		(*******************************************************************************
		  Modify error 
		********************************************************************************)
		E_ITC_MsgTypeConv.E_ERROR_REQUEST:
			M_ITC_ERQ(meChannelSrc := meChannelSrc, mpData := mpData, mLen := mLen);

	ELSE
		// Unknown ITC message type received
		DebugMsg := CONCAT('Subsystem emulation unknown ITC Message type: ', INT_TO_STRING(SubsystemBase.eITC_MsgType));
		fbDebugMsg.M_SendErrorMsg(DebugMsg);
	END_CASE

END_IF
END_METHOD

METHOD M_UpdateRealObjectData
(**************************************************************************************
 * 	Application		:	BoxControl Framework
 *	Revision		:	$Revision: 404529 $
 *	Revision date	:	$Date: 2018-04-23 08:21:38 +0200 (Mo., 23 Apr 2018) $
 *	Last changed by	:	$Author: b7bolm $
 *	URL				:	$URL: http://almscdc.swisslog.com/repo/SWPD/Development/BoxControlFramework/20_Release/trunk/01_Software/BCF/BCF/JumpStart/20_Product/11_Emu/15_Subsystem/10_Lib/10_Conv/FB_SubsystemConvEmulation.TcPOU $
 *
 *	Purpose			:	This methode gets always the current values of the real object
 *
 * ------------------------------------------------------------------------------------
 *	Copyright Swisslog [IP AG], Switzerland. All rights reserved.
 * 
 * ------------------------------------------------------------------------------------
 *	
 * 	Revision History: 
 *
 * 	VERSION			DATE			INITIALS			DESCRIPTION
 *	0.1				01.01.2001		swl					Example
 *
 **************************************************************************************)

IF __ISVALIDREF(SubsystemRegistry.rSubsystemData) THEN
	SubsystemBase.rSubsystemDataReal REF= SubsystemRegistry.rSubsystemData;
ELSE
	SubsystemBase.rSubsystemDataReal REF= SubsystemBase.SubsystemDataEmpty;
END_IF

IF __ISVALIDREF(SubsystemRegistry.rSubsystemInterface) THEN
	SubsystemBase.rSubsystemInterfaceReal REF= SubsystemRegistry.rSubsystemInterface;
ELSE
	SubsystemBase.rSubsystemInterfaceReal REF= SubsystemBase.SubsystemInterfaceEmpty;
END_IF

IF __ISVALIDREF(SubsystemRegistry.rSettingsSubsystem) THEN
	SubsystemBase.rSettingsSubsystemReal REF= SubsystemRegistry.rSettingsSubsystem;
ELSE
	SubsystemBase.rSettingsSubsystemReal REF= SubsystemBase.SettingsSubsystemEmpty;
END_IF
END_METHOD

END_FUNCTION_BLOCK

// ---- 20_Product/10_BCF/10_Base/11_Com/12_DebugMsg/FB_DebugMsgManager.TcPOU
{attribute 'reflection' := ''}
FUNCTION_BLOCK FB_DebugMsgManager
(**************************************************************************************
 * 	Application		:	BoxControl Framework
 *	Revision		:	$Revision: 404529 $
 *	Revision date	:	$Date: 2018-04-23 08:21:38 +0200 (Mo., 23 Apr 2018) $
 *	Last changed by	:	$Author: b7bolm $
 *	URL				:	$URL: http://almscdc.swisslog.com/repo/SWPD/Development/BoxControlFramework/20_Release/trunk/01_Software/BCF/BCF/JumpStart/20_Product/10_App/11_Com/10_Lib/FB_DebugMsgManager.TcPOU $
 *
 *	Purpose			:	Debug msg manager 
 *
 * ------------------------------------------------------------------------------------
 *	Copyright Swisslog [IP AG], Switzerland. All rights reserved.
 * 
 * ------------------------------------------------------------------------------------
 *	
 * 	Revision History: 
 *
 * VERSION DATE         INITIALS     DESCRIPTION
 * 0.0     DD.MM.YYYY   (name)       (explain customized modifications)
 *
 **************************************************************************************)
VAR_INPUT
	Config						: ST_CFG_DebugMsgManager;	// Configuration of debug msg manager
	//-----------------------------------------------------------------------------------
	EnableInfos					: BOOL		:= TRUE;		// Enables debug messages for infos
	EnableWarnings				: BOOL		:= TRUE;		// Enables debug messages for warnings
	EnableErrors				: BOOL		:= TRUE;		// Enables debug messages for errors
END_VAR
 
VAR
	DebugMsg					: T_MaxString; // String to compose the logmessage
	fbDebugMsg					: FB_DebugMsg; // Object Debug instance
	fbTCP_Driver				: FB_TCP_Driver; // Instance of a TCP/IP connection handler
	AddByteMessage				: ARRAY[1 .. MAX_MSG_LENGTH] OF BYTE; // Added byte message
	ReadByteMessage				: ARRAY[1 .. MAX_MSG_LENGTH] OF BYTE; // Read out message
	CollectedByteMessage		: ARRAY[1 .. MAX_MSG_LENGTH] OF BYTE; // Collected byte message
	SendBufferSpace				: ARRAY[1 .. MAX_BUFFER_SPACE] OF BYTE; // Space for send messages
	fbSendBuffer				: FB_MemRingBuffer; // Send buffer
	Header						: T_MaxString; // Collected header
	LastAddedMsg				: T_MaxString; // Debug message last added message
	LastSentMsg					: T_MaxString; // Debug message last sent
	WritePointer				: UDINT; // Counter for assembling byte stream
	NoError						: BOOL; // No error during operation
	DataReady					: BOOL; // Data ready to send
	Idx							: INT; // Index for iteration	
	RecvData					: ARRAY[1..10] OF BYTE; // Receive buffer
	fbFileHandler				: FB_TraceHandler(); 					// trace file handler
END_VAR

VAR CONSTANT
	MAX_MSG_LENGTH				: DINT := 30000; // Maximum byte length of a message
	MAX_BUFFER_SPACE			: DINT := 30000; // Allocated send buffer space
	MSG_PER_CYCLE				: INT := 5; // Maximum collected messages
	DEBUGMESSAGETYPELENGTH 		: INT := 20; // String length debug message type
END_VAR


// call file handler
fbFileHandler();

// Only handle all entries, if a connection is established
IF fbTCP_Driver.Connected THEN
	// Check if a message to send is available and the sending channel is free to send
	IF NOT fbTCP_Driver.SendBusy AND fbSendBuffer.nCount > 0 THEN
			
		// Initialize values
		MEMSET(destAddr := ADR(CollectedByteMessage), 0, SIZEOF(CollectedByteMessage));
		WritePointer := 0;
		DataReady := FALSE;
		(*
		In order to send efficiently, it will be tried to collect
		multiple messages to one TCP/IP stream.
		
		Generell it will be tried to collect everytime MSG_PER_CYCLE messages.
		After MSG_PER_CYCLE messages or if the added messages exeeds MAX_MSG_LENGTH, 
		no more messages will be added.
		*)
		FOR Idx := 1 TO MSG_PER_CYCLE DO
			// If send buffer consists of unsent messages
			IF fbSendBuffer.nCount > 0 THEN
				// Clear byte stream
				MEMSET(destAddr := ADR(ReadByteMessage), 0, SIZEOF(ReadByteMessage));
				
				// Read next message out of the buffer (But not remove)
				fbSendBuffer.A_GetHead(
					pBuffer := ADR(SendBufferSpace), 
					cbBuffer := SIZEOF(SendBufferSpace), 
					pRead := ADR(ReadByteMessage), 
					cbRead := SIZEOF(ReadByteMessage));
				
				// If read out was successfully
				IF fbSendBuffer.bOk THEN
					// Append source
					NoError := F_AssembleByteStream(
									pSrc := ADR(ReadByteMessage), 
									SrcLen := fbSendBuffer.cbReturn,
									pDest := ADR(CollectedByteMessage), 
									DestLen := SIZEOF(CollectedByteMessage),
									WritePointer := WritePointer);
					
					// if assembling was successful (Maybe the message was to long and therefore not adable
					IF NoError THEN
						// As a reason that the message could be assembled, remove from buffer
						fbSendBuffer.A_RemoveHead(
							pBuffer := ADR(SendBufferSpace), 
							cbBuffer := SIZEOF(SendBufferSpace), 
							pRead := ADR(ReadByteMessage), 
							cbRead := SIZEOF(ReadByteMessage));
							
						// Data assembled
						DataReady := TRUE;
					ELSE
						(*
						It was not possible to add MSG_PER_CYCLE messages.
						Already added messages exeeded MAX_MSG_LENGTH
						*)
						EXIT;
					END_IF	
				ELSE
					DebugMsg := CONCAT('CRITICAL Buffer read out. ReturnValue:', UDINT_TO_STRING(fbSendBuffer.cbReturn));
					fbDebugMsg.M_SendErrorMsg(DebugMsg);	
				END_IF
			ELSE
				// No further messages waiting
				EXIT;
			END_IF
		END_FOR
	
		// If data needs to be sent
		IF DataReady THEN
			// Send command
			fbTCP_Driver.M_Send(
				mpSendData	:= ADR(CollectedByteMessage),
				mSendDataLen:= WritePointer);
				
			// Store first 255 characters for debugging
			F_BlockCopy(
				pSrc:= ADR(CollectedByteMessage), 
				LenSrc:= WritePointer, 
				pDest:= ADR(LastSentMsg), 
				LenDest:= SIZEOF(LastSentMsg));
		END_IF
	END_IF
END_IF

// Cylic update of TCP/ IP driver
// Receive is not needed for debug messages, therefore no receive structure is allocated
// Call is at the end, to gain one cycle of a sending request
fbTCP_Driver(
	Config := Config.TCP_Driver, 
    pReceiveData := ADR(RecvData),
	ReceiveDataLen := SIZEOF(RecvData));

// file handler
{attribute 'monitoring' := 'call'}
PROPERTY PUBLIC FileHandler : I_TraceHandler
GET
FileHandler:= fbFileHandler;
END_GET
END_PROPERTY

{attribute 'object_name' := 'M_SendMessage'}
METHOD M_SendMessage : BOOL
(**************************************************************************************
 * 	Application		:	BoxControl Framework
 *	Revision		:	$Revision: 404529 $
 *	Revision date	:	$Date: 2018-04-23 08:21:38 +0200 (Mo., 23 Apr 2018) $
 *	Last changed by	:	$Author: b7bolm $
 *	URL				:	$URL: http://almscdc.swisslog.com/repo/SWPD/Development/BoxControlFramework/20_Release/trunk/01_Software/BCF/BCF/JumpStart/20_Product/10_App/11_Com/10_Lib/FB_DebugMsgManager.TcPOU $
 *
 *	Purpose			:	Send  message
 *
 * ------------------------------------------------------------------------------------
 *	Copyright Swisslog [IP AG], Switzerland. All rights reserved.
 * 
 * ------------------------------------------------------------------------------------
 *	
 * 	Revision History: 
 *
 * 	VERSION			DATE			INITIALS			DESCRIPTION
 *	0.1				01.01.2001		swl					Example
 *
 **************************************************************************************)
VAR_INPUT
	meMessageType		: E_DebugMsgType;
	mDebugSource		: STRING(DEBUGSOURCELENGTH);
	mpMsgData			: PVOID; // Address to the send data storage
	mMsgDataLen			: UDINT; // Data length which need to be sent
END_VAR

VAR
	mString				:STRING(10); // Temp String
END_VAR

// forward to file handler
fbFileHandler.Put(MsgType :=     meMessageType,
                  Instance:= ADR(mDebugSource),
                  Text    :=     mpMsgData);


// Translate to string
CASE meMessageType OF
E_DebugMsgType.INFO:		IF NOT EnableInfos		THEN  M_SendMessage:= FALSE;  RETURN;  END_IF
E_DebugMsgType.WARNING:		IF NOT EnableWarnings	THEN  M_SendMessage:= FALSE;  RETURN;  END_IF
E_DebugMsgType.ERROR:		IF NOT EnableErrors		THEN  M_SendMessage:= FALSE;  RETURN;  END_IF
ELSE						meMessageType:= E_DebugMsgType.ERROR;
END_CASE


// Reset
MEMSET(destAddr := ADR(AddByteMessage), 0, SIZEOF(AddByteMessage));
WritePointer := 0;

Header := CONCAT('<', TimeStampString);
Header := CONCAT(Header, ', ');
Header := CONCAT(Header, TO_STRING(meMessageType));
Header := CONCAT(Header, ', System: ');
Header := CONCAT(Header, INT_TO_STRING(Config.SystemNumber));
Header := CONCAT(Header, ', ');
Header := CONCAT(Header, mDebugSource);
Header := CONCAT(Header, ', ');

// Append header
F_AssembleByteStream(
	pSrc := ADR(Header),
	SrcLen := INT_TO_UDINT(LEN(Header)),
	pDest := ADR(AddByteMessage), 
	DestLen := SIZEOF(AddByteMessage),
	WritePointer := WritePointer);

// Append message
F_BlockCopy(
	pSrc := mpMsgData,
	LenSrc := mMsgDataLen, 
	pDest := ADR(AddByteMessage) + WritePointer,
	LenDest := SIZEOF(AddByteMessage) - WritePointer);

// Update pointer
WritePointer := WritePointer + mMsgDataLen;

// Append end sign + Line feed
mString := '>$0A';

F_AssembleByteStream(
	pSrc := ADR(mString), 
	SrcLen := INT_TO_UDINT(LEN(mString)),
	pDest := ADR(AddByteMessage), 
	DestLen := SIZEOF(AddByteMessage),
	WritePointer := WritePointer);


// Add to byte buffer in order to release caller
fbSendBuffer.A_AddTail(
	pBuffer := ADR(SendBufferSpace), 
	cbBuffer := SIZEOF(SendBufferSpace), 
	pWrite := ADR(AddByteMessage), 
	cbWrite := WritePointer);

IF NOT fbSendBuffer.bOk THEN
	// Remove oldest entry
	fbSendBuffer.A_RemoveHead(
		pBuffer := ADR(SendBufferSpace), 
		cbBuffer := SIZEOF(SendBufferSpace), 
		pRead := ADR(ReadByteMessage), 
		cbRead := SIZEOF(ReadByteMessage));

	// Add to byte buffer in order to release caller
	fbSendBuffer.A_AddTail(
		pBuffer := ADR(SendBufferSpace), 
		cbBuffer := SIZEOF(SendBufferSpace), 
		pWrite := ADR(AddByteMessage), 
		cbWrite := WritePointer);
END_IF

// Store first 255 characters for debugging
F_BlockCopy(
	pSrc:= ADR(AddByteMessage), 
	LenSrc:= WritePointer, 
	pDest:= ADR(LastAddedMsg), 
	LenDest:= SIZEOF(LastAddedMsg));
	
// Return result
M_SendMessage := fbSendBuffer.bOk;
END_METHOD

END_FUNCTION_BLOCK

// ---- 20_Product/30_Toolbox/11_Com/10_TCP_Driver/FB_TCP_Driver.TcPOU
///TCP / IP Driver - Handles a connection to one partner. Handles only one incoming and one outgoing message at once.
FUNCTION_BLOCK FB_TCP_Driver
(**************************************************************************************
* Application : BoxControl Framework 
* Revision date : $Date: 2020-10-16 11:02:56 +0200 (fre, 16 okt 2020) $
* Author : CDC
* ------------------------------------------------------------------------------------ 
* © Swisslog AG 
* Swisslog is not liable for any usage of this source code that is not agreed 
* on between Swisslog and the other party. The mandatory legal liability remains 
* unaffected. 
* ------------------------------------------------------------------------------------ 
* Project revision history: 
* 
* VERSION 	DATE 		INITIALS 	DESCRIPTION 
* 0.1 		12.10.2020 	swl. 		example
* 
**************************************************************************************)

VAR_INPUT
	Config						: ST_CFG_TcpDriver;
	pReceiveData				: PVOID; // Pointer to receive structure
	ReceiveDataLen				: UDINT; // Length of received structure (Maximum which could be received)

END_VAR

VAR_OUTPUT
	NewData						: BOOL; // New Data received	
	ReceivedBytes				: UDINT; // Amount of received bytes
	Connected					: BOOL; // Connected 
	
	ConnBusy					: BOOL; // Connection ongoing
	ConnError					: BOOL; // Error during connection
	ConnErrId					: UDINT; // Connection error code
		
	SendBusy					: BOOL; // Send ongoing status	
	SendError					: BOOL; // Send error
	SendErrId					: UDINT; // Sending error code
	
	RecvBusy					: BOOL; // Receive ongoing status
	RecvError					: BOOL; // Receive error
	RecvErrId					: UDINT; // Receive error code
END_VAR

VAR

	Init						: BOOL := FALSE; // Instance is initialized
	fbDebugMsg					: FB_DebugMsg; // Debug msg handler
	DebugMsg					: T_MAXSTRING; // Debug msg
	EnableSystemLog				: BOOL	:= FALSE;

	fbConnectClientServer		: FB_ClientServerConnection := (sSrvNetId := ''); // Tc library connect
	fbConnectServerClient		: FB_ServerClientConnection; // Tc library connect
	
	fbSocketSend				: FB_SocketSend := (sSrvNetID := '', tTimeout := DEFAULT_ADS_TIMEOUT); // Tc library send
	fbSocketReceive				: FB_SocketReceive := (sSrvNetID := '', tTimeout := DEFAULT_ADS_TIMEOUT); // Tc library recv
	hServer						: T_HSERVER; // Server connection handle 
	hSocket						: T_HSOCKET; // Connection socket
	
	// Send receive data
	RecvString					: T_MaxString; // String received for debugging
	SendString					: T_MaxString; // String send for debugging
	pSendData					: PVOID; // Address send structure
	SendDataLen					: UDINT; // Send data length
	
	// States	
	SocketState					: E_SocketConnectionState := eSOCKET_DISCONNECTED; // TCP/IP connection state 
	ConnState					: E_ConnStates; // Connection states
	SendState					: E_SendStates; // Sending states
	RecvState					: E_RecvStates; // Receive states

	SendTrigger					: BOOL; // New Data to Send
	RestartCom					: BOOL; // Close and reopen socket

	// Socket variables to accept and refuse a second server connection 
	fbConnectServer_ConRefuse	: FB_ServerClientConnection; // Establishes a connection 
	hSocket_ConRefuse			: T_HSOCKET; // Socket handle for this connection
	SocketState_ConRefuse		: E_SocketConnectionState := eSOCKET_DISCONNECTED; // Socket state

	ConnState_ConRefuse			: E_ConnStates; // Connection states; 

	fbSocketSend_ConRefuse		: FB_SocketSend := (sSrvNetID := '', tTimeout := DEFAULT_ADS_TIMEOUT); // Send function block
	MsgConnection_ConRefuse		: STRING := 'Connection refused'; // 

END_VAR

(**************************************************************************************
   		Initialize
***************************************************************************************)

M_Init(FALSE);

//  Server mode
IF Config.Server THEN
	// Call connection handling as server
	A_Server();
	
	// Reject additional incomming connection requests
	A_RejectCon();
	
// Client mode	
ELSE
	// Call connection handling as client
	A_Client();
END_IF

ACTION A_Client:
fbConnectClientServer(hSocket => hSocket);

// Connection states
CASE ConnState OF
	// Connection is idle 
	E_ConnStates.CONN_IDLE:
		Connected := FALSE;
		// If connection is enabled 
		IF Config.EnableConnection THEN
			// Poll connection for new client
			fbConnectClientServer( 	
						nMode			:= SEL( EnableSystemLog, 0, CONNECT_MODE_ENABLEDBG), // Enable/disable debug messages? 
						sRemoteHost 	:= Config.RemoteHost, 
						nRemotePort 	:= Config.RemotePort,
						bEnable			:= TRUE, 
						tReconnect		:= Config.ClientRetryInterval, // Retry connection after  ConnectionTimeout
						eState			=> SocketState );
						
			IF NOT fbConnectClientServer.bBusy THEN
				IF NOT fbConnectClientServer.bError THEN
					IF SocketState = eSOCKET_CONNECTED THEN  // We are connected 
											
						SendBusy 	:= FALSE;
						RecvBusy 	:= FALSE;
	
						Connected := TRUE;
						ConnState := E_ConnStates.CONN_RUNNING;
					END_IF
				END_IF
			END_IF				
		
		END_IF
		

	// Connection is established - execute sending and receive over the connection 
	E_ConnStates.CONN_RUNNING:
		// Send
		A_Send();
		// Recv
		A_Recv();

	
		// Should the connection need to be disabled or an error occours in the sending/receiving of data, deal with it 
		IF NOT Config.EnableConnection AND NOT fbSocketSend.bBusy AND NOT fbSocketReceive.bBusy OR RestartCom THEN
			RestartCom := FALSE;
			M_DebugSendInfoMsg('ConnState: CONN_CLOSE_START');
			ConnState := E_ConnStates.CONN_CLOSE;
			
		ELSIF SendError OR RecvError THEN
			SendError := FALSE;
			RecvError := FALSE;
			M_DebugSendInfoMsg('ConnState: CONN_ERROR');
			ConnState := E_ConnStates.CONN_ERROR;
		END_IF
		
	// Connections need to be closed 
	E_ConnStates.CONN_CLOSE:
		fbConnectClientServer( bEnable:= FALSE, eState => SocketState );
		IF SocketState = eSOCKET_DISCONNECTED THEN
			// Please wait some seconds and then try to connect again 
			Connected := FALSE;
			RecvState := E_RecvStates.RECV_IDLE;
			SendState := E_SendStates.SEND_IDLE;
			ConnState := E_ConnStates.CONN_IDLE;
		END_IF
		
	// Error detected in connection 
	E_ConnStates.CONN_ERROR:
		
		// If still connected
		IF Connected THEN
			// Close connection
			M_DebugSendInfoMsg('ConnState: CONN_CLOSE_START');
			ConnState := E_ConnStates.CONN_CLOSE;
		ELSE
			ConnBusy   := FALSE;
			// Switch to idle
			M_DebugSendInfoMsg('ConnState: CONN_IDLE');
			ConnState := E_ConnStates.CONN_IDLE;
		END_IF
END_CASE
END_ACTION

ACTION A_Recv:
// Receive states
CASE RecvState OF
	// Idle state - waiting for confirmation to enable receiving 
	E_RecvStates.RECV_IDLE:
		// If no new data are waiting to be removed and
		// a valid receive structure is available
		IF NOT NewData AND
           pReceiveData <> 0 AND 
           ReceiveDataLen > 0 THEN
			// Block receive channel
			RecvBusy := TRUE;
			
			// Call receive function block
			fbSocketReceive(
				hSocket  	:= hSocket,
				pDest	 	:= pReceiveData,
				cbLen	 	:= ReceiveDataLen,
				bExecute 	:= TRUE);
			
			// Reset variables
			RecvError := FALSE;
			RecvErrId := 0;
			ReceivedBytes := 0;
			MEMSET(ADR(RecvString), 0, SIZEOF(RecvString));
			
			// Switch to receive start
			RecvState := E_RecvStates.RECV_WAIT;
		
		END_IF
		
	// Receiving is active, wait for the function to complete 
	E_RecvStates.RECV_WAIT:
		// Reset
		fbSocketReceive(bExecute := FALSE);
		
		// If receiving is finished
		IF NOT fbSocketReceive.bBusy THEN
			// Reset
			RecvBusy := FALSE;	
		
			// If no error is occured
			IF NOT fbSocketReceive.bError THEN
				// Receive module has completed - analyse the message 
				IF (fbSocketReceive.nRecBytes > 0) THEN
					// Store received bytes 
					ReceivedBytes := fbSocketReceive.nRecBytes;
				
					// Copy first 255 signs for debug reason to RecvString
					F_BlockCopy(
						pSrc:= pReceiveData, 
						LenSrc:= ReceivedBytes, 
						pDest:= ADR(RecvString), 
						LenDest:= SIZEOF(RecvString));
						
					// Set new data ready
					NewData := TRUE;
				END_IF
				// Go to Idle
				RecvState := E_RecvStates.RECV_IDLE;
			ELSE
				// Error detected 
				RecvErrId := fbSocketReceive.nErrId;
				RecvState := E_RecvStates.RECV_ERROR;
			END_IF
		END_IF
		
	// Recv error state 
	E_RecvStates.RECV_ERROR:
		RecvBusy := FALSE;
		RecvError := TRUE;
		RecvState := E_RecvStates.RECV_IDLE;
END_CASE
END_ACTION

ACTION A_RejectCon:
(* -----------------------------------------------------------------------------
 	This code avoids addional connection as soon as a connection was established
 	It will accept any new incomming connection requests and will close it immediately
-------------------------------------------------------------------------------- *)

// Connection alreads established check for new incomming connection requests
IF ConnState <> E_ConnStates.CONN_IDLE THEN

	// Connection states
	CASE ConnState_ConRefuse OF
		// Connection is idle 
		E_ConnStates.CONN_IDLE:
			
			// If connection is enabled and not listening
			IF Config.EnableConnection THEN
				fbConnectServer_ConRefuse( 	eMode := eACCEPT_ALL, 
								tReconnect := Config.ServerRetryInterval, // Retry connection after  ConnectionTimeout
								bEnable := TRUE, 
								hServer := hServer, 
								hSocket => hSocket_ConRefuse, 
								eState => SocketState_ConRefuse );
								
				IF NOT fbConnectServer_ConRefuse.bBusy THEN
					IF NOT fbConnectServer_ConRefuse.bError THEN
						IF SocketState = eSOCKET_CONNECTED THEN(* We are connected *)
							ConnState_ConRefuse := E_ConnStates.CONN_RUNNING;
						END_IF
					END_IF
				END_IF
			END_IF
	
		// Socket is open and listening, process incoming connection requests from partner 
		E_ConnStates.CONN_RUNNING:
					
			// Start send action in same cycle
			MsgConnection_ConRefuse := 'Connection refused, already active Connection with IP = ';
			MsgConnection_ConRefuse := concat(MsgConnection_ConRefuse, fbConnectServerClient.hSocket.remoteAddr.sAddr);

			// Send the connection refused message to the client
			fbSocketSend_ConRefuse(
				hSocket  	:= hSocket_ConRefuse,
				pSrc     	:= ADR(MsgConnection_ConRefuse),
				cbLen    	:= SIZEOF(MsgConnection_ConRefuse),
				bExecute 	:= TRUE);
					
					
			// Continue to wait, until the FB_SocketSend instance has finished and close the connection
			IF NOT fbSocketSend_ConRefuse.bBusy THEN
				// Reset
				MsgConnection_ConRefuse := '';
				fbSocketSend_ConRefuse(
					hSocket  	:= hSocket_ConRefuse,
					pSrc     	:= ADR(MsgConnection_ConRefuse),
					cbLen    	:= SIZEOF(MsgConnection_ConRefuse),
					bExecute 	:= FALSE);
			
				ConnState_ConRefuse := E_ConnStates.CONN_CLOSE;
			END_IF
					
		// Close the socket 
		E_ConnStates.CONN_CLOSE:
					
			fbConnectServer_ConRefuse( hServer := hServer, bEnable:= FALSE, eState => SocketState_ConRefuse );
			// Socket closed
			IF SocketState_ConRefuse = eSOCKET_DISCONNECTED THEN
				ConnState_ConRefuse := E_ConnStates.CONN_IDLE;
			END_IF
	
	END_CASE

// Disable listener for additional connection requests, active connection was closes 	
ELSE
	fbConnectServer_ConRefuse(
						hServer := hServer,  
						bEnable := FALSE); 
END_IF
END_ACTION

ACTION A_Send:
CASE SendState OF
		// Idle State - Waiting for trigger to start sending 
		E_SendStates.SEND_IDLE:
			// When new data are ready to be sent
			// and an valid send structure is available
			IF SendTrigger AND
			   pSendData > 0 AND 
			   SendDataLen > 0 THEN
			   	// Block send channel
				SendBusy    := TRUE;
				
				// Copy first 255 signs for debug reason to SendString
				F_BlockCopy(
					pSrc:= pSendData, 
					LenSrc:= SendDataLen, 
					pDest:= ADR(SendString), 
					LenDest:= SIZEOF(SendString));
				
				// Start send action in same cycle
				fbSocketSend(
					hSocket  	:= hSocket,
					pSrc     	:= pSendData,
					cbLen    	:= SendDataLen,
					bExecute 	:= TRUE);
				
				// Reset variables
				SendError   := FALSE;
				SendErrId   := 0;
				
				SendState  := E_SendStates.SEND_WAIT;
			ELSIF SendTrigger THEN 
				//If for some reason the data gets reset while send trigger is on and there is an error, the send will get stuck, so lets reset the send trigger.
				SendTrigger := FALSE;
				
				DebugMsg := CONCAT('Send trigger on while there is no data present. SendDataLen: ', UDINT_TO_STRING(SendDataLen));
				fbDebugMsg.M_SendWarningMsg(DebugMsg);
			END_IF
				
		// Data has been queued for sending. Wait to see if sending was successful. 
		E_SendStates.SEND_WAIT:
			fbSocketSend(bExecute := TRUE);
			// Continue to wait, until the FB_SocketSend instance has finished
			IF NOT fbSocketSend.bBusy THEN
				// Reset
				SendBusy := FALSE;
				fbSocketSend(bExecute := FALSE);
				
				IF NOT fbSocketSend.bError THEN
					SendTrigger := FALSE;
					// Sending completed without error, return to sending idle state and wait for next message to send 
					SendState 	:= E_SendStates.SEND_IDLE;
				ELSE
					// Error detected 
					SendErrId := fbSocketSend.nErrId;
					SendState := E_SendStates.SEND_ERROR;
				END_IF
			END_IF
			
		// Send error state 
		E_SendStates.SEND_ERROR:
			SendBusy := FALSE;
			SendError := TRUE;
			SendState := E_SendStates.SEND_IDLE;
	END_CASE
END_ACTION

ACTION A_Server:
fbConnectServerClient(hServer := hServer,
				hSocket => hSocket, 
				eState => SocketState );
					  
					  
// Connection states
CASE ConnState OF
	// Connection is idle 
	E_ConnStates.CONN_IDLE:
		// Reset
		Connected := FALSE;
		
		// If connection is enabled and not listning
		IF Config.EnableConnection THEN
			fbConnectServerClient( 	eMode := eACCEPT_ALL, 
							tReconnect := Config.ServerRetryInterval, // Retry connection after  ConnectionTimeout
							bEnable := TRUE, 
							hServer := hServer, 
							eState => SocketState );
							
			IF NOT fbConnectServerClient.bBusy THEN
				IF NOT fbConnectServerClient.bError THEN
					IF SocketState = eSOCKET_CONNECTED THEN(* We are connected *)
						
						SendBusy := FALSE;
						RecvBusy := FALSE;
	
						// Connected
						Connected := TRUE;
						ConnState := E_ConnStates.CONN_RUNNING;
					END_IF
				END_IF
			END_IF
		END_IF
		
		
	// Socket is open and listening, process incoming connection requests from partner 
	E_ConnStates.CONN_RUNNING:

			// Send
			A_Send();
			// Recv
			A_Recv();

		
		// Should the connection need to be disabled or an error occours in the Sending/Receiving of data, deal with it 
		IF NOT Config.EnableConnection AND NOT fbSocketSend.bBusy AND NOT fbSocketReceive.bBusy OR RestartCom THEN
			RestartCom := FALSE;
			M_DebugSendInfoMsg('AcceptState: ACCEPT_CLOSE_START');
			ConnState := E_ConnStates.CONN_CLOSE;
		ELSIF SendError OR RecvError THEN
			SendError := FALSE;
			RecvError := FALSE;
			M_DebugSendInfoMsg('AcceptState: ACCEPT_ERROR');
			ConnState := E_ConnStates.CONN_ERROR;
		END_IF
				
	// Close the socket 
	E_ConnStates.CONN_CLOSE:
				
		fbConnectServerClient( hServer := hServer, bEnable:= FALSE, eState => SocketState );
		IF SocketState = eSOCKET_DISCONNECTED THEN
			Connected := FALSE;
			RecvState := E_RecvStates.RECV_IDLE;
			SendState := E_SendStates.SEND_IDLE;				
			ConnState := E_ConnStates.CONN_IDLE;
		END_IF
		
	// Error state 
	E_ConnStates.CONN_ERROR:
		
		// If still connected
		IF Connected THEN
			// Close connection
			M_DebugSendInfoMsg('ConnState: CONN_CLOSE_START');
			ConnState := E_ConnStates.CONN_CLOSE;
		ELSE
			ConnBusy   := FALSE;
			// Switch to idle
			M_DebugSendInfoMsg('ConnState: CONN_IDLE');
			ConnState := E_ConnStates.CONN_IDLE;
		END_IF		
END_CASE
END_ACTION

METHOD M_DataProcessed
// Release receive channel
NewData := FALSE;
END_METHOD

METHOD PRIVATE M_DebugSendInfoMsg
(**************************************************************************************
 * 	Application		:	BoxControl Framework
 *	Revision		:	$Revision: 404529 $
 *	Revision date	:	$Date: 2020-10-16 11:02:56 +0200 (fre, 16 okt 2020) $
 *	Last changed by	:	$Author: b7bolm $
 *	URL				:	$URL: http://almscdc.swisslog.com/repo/SWPD/Development/BoxControlFramework/20_Release/trunk/01_Software/BCF/BCF/JumpStart/30_Toolbox/11_Com/10_TCP_Driver/FB_TCP_Driver.TcPOU $
 *
 *	Purpose			:	Send debug message, needs to enabable via TCP-Configuration
 *
 *
 * ------------------------------------------------------------------------------------
 *	Copyright Swisslog [IP AG], Switzerland. All rights reserved.
 * 
 * ------------------------------------------------------------------------------------
 *	
 * 	Revision History: 
 *
 * 	VERSION			DATE			INITIALS			DESCRIPTION
 *	0.1				01.01.2001		swl					Example
 *
 **************************************************************************************)
VAR_INPUT
	mDebugMessage: STRING(DEBUGMESSAGELENGTH);
END_VAR
IF Config.EnableDebugMsg THEN
	fbDebugMsg.M_SendInfoMsg(mDebugMessage);
END_IF
END_METHOD

{attribute 'object_name' := 'M_Init'}
METHOD M_Init
(**************************************************************************************
 * 	Application		:	BoxControl Framework
 *	Revision		:	$Revision: 404529 $
 *	Revision date	:	$Date: 2020-10-16 11:02:56 +0200 (fre, 16 okt 2020) $
 *	Last changed by	:	$Author: b7bolm $
 *	URL				:	$URL: http://almscdc.swisslog.com/repo/SWPD/Development/BoxControlFramework/20_Release/trunk/01_Software/BCF/BCF/JumpStart/30_Toolbox/11_Com/10_TCP_Driver/FB_TCP_Driver.TcPOU $
 *
 *	Purpose			:	Initialize TCP/ Ip Driver.
 *						Normal calling will only do a init if its needed. If this 
 *						instance is called with mInit = TRUE, initialization is forced
 *
 * ------------------------------------------------------------------------------------
 *	Copyright Swisslog [IP AG], Switzerland. All rights reserved.
 * 
 * ------------------------------------------------------------------------------------
 *	
 * 	Revision History: 
 *
 * 	VERSION			DATE			INITIALS			DESCRIPTION
 *	0.1				01.01.2001		swl					Example
 *
 **************************************************************************************)
VAR_INPUT
	mInit				: BOOL; // Force initialization
END_VAR
// Check if init is requested or needed
IF NOT Init OR mInit THEN
	IF Config.EnableConnection THEN
		// Init done
		Init := TRUE;

		// Initialize bits
		Connected		:= FALSE;
		ConnBusy 		:= FALSE;
		ConnError		:= FALSE;
		ConnErrId		:= 0;
		SendBusy		:= FALSE;
		SendError		:= FALSE;
		SendErrId		:= 0;
		RecvBusy		:= FALSE;
		RecvError		:= FALSE;
		RecvErrId		:= 0;
		ReceivedBytes   := 0;
	
		// Close all channels - and do a connection retry
		ConnState := E_ConnStates.CONN_CLOSE;
		
		IF Config.Server THEN
			// Initialize server handle once 
			IF NOT F_CreateServerHnd( 	sSrvNetID := '', 
								sLocalHost := Config.LocalHost, 
								nLocalPort	:= Config.LocalPort,
//								nMode 		:= SEL( EnableSystemLog, 0, CONNECT_MODE_ENABLEDBG OR LISTEN_MODE_CLOSEALL),(* Enable/disable debug messages? *)
								nMode 		:= SEL( EnableSystemLog, 0, CONNECT_MODE_ENABLEDBG),(* Enable/disable debug messages? *)
								bEnable 	:= FALSE,(* TRUE = leave listener socket open, FALSE = close listener socket after last connection ist closed too *)
								hServer 	:= hServer ) THEN
	
				// Init failed server handle is not valid
				Init := FALSE;
				M_DebugSendInfoMsg('Init: Server handle not valid');				
			END_IF				
	
		END_IF
	END_IF	
END_IF
END_METHOD

{attribute 'object_name' := 'M_RestartCom'}
METHOD M_RestartCom
(**************************************************************************************
 * 	Application		:	BoxControl Framework
 *	Revision		:	$Revision: 404529 $
 *	Revision date	:	$Date: 2020-10-16 11:02:56 +0200 (fre, 16 okt 2020) $
 *	Last changed by	:	$Author: b7bolm $
 *	URL				:	$URL: http://almscdc.swisslog.com/repo/SWPD/Development/BoxControlFramework/20_Release/trunk/01_Software/BCF/BCF/JumpStart/30_Toolbox/11_Com/10_TCP_Driver/FB_TCP_Driver.TcPOU $
 *
 *	Purpose			:	Restart TCP/IP Driver.
 *
 *
 * ------------------------------------------------------------------------------------
 *	Copyright Swisslog [IP AG], Switzerland. All rights reserved.
 * 
 * ------------------------------------------------------------------------------------
 *	
 * 	Revision History: 
 *
 * 	VERSION			DATE			INITIALS			DESCRIPTION
 *	0.1				01.01.2001		swl					Example
 *
 **************************************************************************************)
M_Init(TRUE);
END_METHOD

METHOD M_Send : BOOL
VAR_INPUT
	mpSendData		: PVOID; // Address to the send data storage
	mSendDataLen	: UDINT; // Data length which need to be sent
END_VAR
// Check inputs
IF mpSendData = 0 OR mSendDataLen = 0 THEN
	M_Send := FALSE;
	RETURN;
END_IF

// If a send request is already waiting or a send process is ongoing -&gt; do nothing
IF SendTrigger OR SendBusy THEN
	M_Send := FALSE;
ELSE
	pSendData := mpSendData;
	SendDataLen := mSendDataLen;
	
	SendTrigger := TRUE;
	
	M_Send := TRUE;
END_IF
END_METHOD

END_FUNCTION_BLOCK

// ---- 20_Product/10_BCF/10_Base/11_Com/12_DebugMsg/20_TraceHandler/FB_TraceHandler.TcPOU
// writes traces into files, deletes too old files and monitors hdd usage
{attribute 'reflection'}
FUNCTION_BLOCK PUBLIC FB_TraceHandler IMPLEMENTS I_TraceHandler
(**************************************************************************************
 *  Application     : BoxControl Framework
 *  Revision        : $Revision: 404529 $
 *  Revision date   : $Date: 2020-10-20 08:21:38 +0200 (Mo., 20 Oct 2020) $
 *  Last changed by : $Author: b7lipim $
 *  URL             : $URL: http://almscdc.swisslog.com/repo/SWPD/Development/BoxControlFramework/20_Release/trunk/01_Software/BCF/BCF/JumpStart/20_Product/10_App/11_Com/10_Lib/FB_DebugMsg.TcPOU $
 *
 *  Purpose :	writes (debug) messages into files in subfolders
 *            deletes all subfolders including files older than 7d (according to name, not date)
 *            monitors hdd usage, reports it via debug message and surpress further writing if 80% is exceeded
 *
 * ------------------------------------------------------------------------------------
 *  Copyright Swisslog [IP AG], Switzerland. All rights reserved.
 * 
 * ------------------------------------------------------------------------------------
 *	
 * 	Revision History: 
 *
 *  VERSION DATE         INITIALS     DESCRIPTION
 *  0.0     DD.MM.YYYY   (name)       (explain customized modifications)
 *
 **************************************************************************************)

(********************************************************************************************************************************)
VAR_STAT CONSTANT
  SHELF_LIFE            : TIME                             := T#7D;      // duration until old folders will be deleted
  (*----------------------------------------------------------------------------------------------------------------------------*)
  MAX_FILEOPEN_TIME     : TIME                             := T#100MS;   // maximum file open time until reopen/flush
  LOCKTIME              : TIME                             := T#100MS;   // inhibit time between write attemts
  (*----------------------------------------------------------------------------------------------------------------------------*)
  BUFFER_SIZE           : WORD                             := 8192;      // size of internal file write buffer
  FIFO_SIZE             : WORD                             := 1024;      // size of internal dynamic fifo to temporary store trace entries
  (*----------------------------------------------------------------------------------------------------------------------------*)
  HDD_WARNING_LEVEL     : BYTE                             := 60;        // warning if hdd usage exceeds this percentage
  HDD_ERROR_LEVEL       : BYTE                             := 80;        // error and stop writing if hdd usage exceeds this percentage
END_VAR

(********************************************************************************************************************************)
VAR
  {attribute 'instance-path'}
  {attribute 'no_init'}
  _Instance             : STRING[255]                      := '';         // instance path
  (*----------------------------------------------------------------------------------------------------------------------------*)
  _Enable               : BOOL                             := FALSE;      // HI = writing/deleting enabled
  _MaxFileSizeKB        : WORD                             := 10_240;     // maximum file size in kilobytes
  _Folder               : A_TracePath                      := '';         // working folder without ending '/'
  (*-- duration ----------------------------------------------------------------------------------------------------------------*)
  _StartSystemTick      : ULINT                            := 0;          // system tick at execution start
  _GetSystemTicks       : GETCPUCOUNTER;                                  // Gets the system time in 100ns ticks  
  (*-- general -----------------------------------------------------------------------------------------------------------------*)
  _GetHostName          : FB_GetHostName()                 := (sNetID:= '', tTimeout:= DEFAULT_ADS_TIMEOUT);
  _GetAdaptersInfo      : FB_GetAdaptersInfo()             := (sNetID:= '', tTimeout:= DEFAULT_ADS_TIMEOUT);
  _GetDeviceIdentificationEx : FB_GetDeviceIdentificationEx:= (sNetID:= '', tTimeout:= DEFAULT_ADS_TIMEOUT);
  _MainFolder           : A_TracePath                      := '';         // working folder ending without '/'
  _Active               : BOOL                             := FALSE;      // HI = enable and working folder exists
  _Opened               : BOOL                             := FALSE;      // HI = file is currently open
  _PlcRestarted         : BOOL                             := TRUE;       // HI = add separation lines to file
  _MillisecondsLast		: WORD                             := 16#FFFF;    // system clock monitoring
  _Text                 : STRING[255]                      := '';         // own debug message
  (*-- checking work folder - states -------------------------------------------------------------------------------------------*)
  _CheckState           : E_TraceCheckStates               := E_TraceCheckStates.Initialization;
  _CheckStateLast       : E_TraceCheckStates               := E_TraceCheckStates.Initialization;
  _CheckTime            : TIME                             := T#0S;
  (*-- writing files - states --------------------------------------------------------------------------------------------------*)
  _WriteState           : E_TraceWriteStates               := E_TraceWriteStates.Initialization;
  _WriteStateLast       : E_TraceWriteStates               := E_TraceWriteStates.Initialization;
  _WriteTime            : TIME                             := T#0S;
  (*-- deleting files - states -------------------------------------------------------------------------------------------------*)
  _DeleteState          : E_TraceDeleteStates              := E_TraceDeleteStates.Initialization;
  _DeleteStateLast      : E_TraceDeleteStates              := E_TraceDeleteStates.Initialization;
  _DeleteTime           : TIME                             := T#0S;
  (*-- hdd monitoring ----------------------------------------------------------------------------------------------------------*)
  _HddUsage             : FB_HddUsage;
  _HddUsageTime         : TIME                             := T#0S;
  _HddUsageCount        : DWORD                            := 0;               // counter
  _HddState             : E_TraceHddUsageStates            := E_TraceHddUsageStates.Initialization;
  _HddStateLast         : E_TraceHddUsageStates            := E_TraceHddUsageStates.Initialization;
  _HddTooFull           : BOOL                             := FALSE;           // hdd is too full to write
  _HddFullMissed        : ULINT                            := 0;               // rejected messages due to hdd too full  ( maybe persistent? )
  (*-- writing files - data ----------------------------------------------------------------------------------------------------*)
  _WritePath            : A_TracePath                      := '';              // current working folder with date and trailing '/'
  _WriteFileName        : A_TracePath                      := '';              // current file name
  _WriteDate            : TIMESTRUCT;                                          // current working date
  (*-- file handling -----------------------------------------------------------------------------------------------------------*)
  _FileSize             : ULINT                            := 0;               // current file size in bytes
  _FileIndex            : WORD                             := 0;               // current file number
  _FileTimeOpened       : TIME                             := T#0S;            // timestamp file was opened
  _CreateDir            : Tc2_System.FB_CreateDir;                             // create new folder
  _FileCheck            : Tc2_Utilities.FB_EnumFindFileEntry;                  // checks current working folder for already existing files
  _FileOpen             : Tc2_System.FB_FileOpen;                              // open/create file
  _FileWrite            : Tc2_System.FB_FileWrite;                             // write into file
  _FileClose            : Tc2_System.FB_FileClose;                             // close file
  (*-- folder handling ---------------------------------------------------------------------------------------------------------*)
  _CheckWorkFolder      : Tc2_Utilities.FB_EnumFindFileEntry;                  // checks working folder being existent
  _ScanSubFolder        : Tc2_Utilities.FB_EnumFindFileEntry;                  // checks current working folder for subfolders
  _FileFind             : Tc2_Utilities.FB_EnumFindFileEntry;                  // checks (old) subfolders for files to delete
  _FileDelete           : Tc2_System.FB_FileDelete;                            // delete file
  _FolderRemove         : Tc2_System.FB_RemoveDir;                             // delete folder
  (*-- write fifo --------------------------------------------------------------------------------------------------------------*)
  _TaskCounter          : WORD                             := 0;               // counter for put calls within one plc cycle
  _FifoFillLevel        : WORD                             := 0;               // fill level
  _FifoInput            : WORD                             := 0;               // (next) input position
  _FifoOutput           : WORD                             := 0;               // (next) output position
  _Fifo                 : ARRAY[0..FIFO_SIZE-1] OF POINTER TO FB_TraceEntry;          // fifo itself
  (*-- write data --------------------------------------------------------------------------------------------------------------*)
  _DataDateChanged      : BOOL                             := FALSE;           // date of write data has changed
  _DataLength           : DWORD                            := 0;               // valid length of _DataBuffer
  _DataBuffer           : ARRAY[0..BUFFER_SIZE-1] OF BYTE;                     // data buffer to write into file
  (*-- diagnostics & statisticals ------------------------------------------------------------------------------------------------*)
  _Statistics           : FB_TraceHandlerStatistics();
  _ExecutionDuration    : ULINT                            := 0;               // duration of execution in microseconds
  _ExecutionNow         : ULINT                            := 0;
  (*-- testing -------------------------------------------------------------------------------------------------------------------*)
  _Diag_SystemTime      : ULINT                            := 0;
  _Diag_NoMemory        : ULINT                            := 0;
  _Diag_NoEntry         : ULINT                            := 0;
  _Diag_FifoFull        : ULINT                            := 0;
  _Diag_InvalidDate     : ULINT                            := 0;
END_VAR

(*****************************************************1*********2*********3*********4*********5*********6*********7*********8****)
VAR_STAT CONSTANT                          // 123456789012345678901234567890123456789012345678901234567890123456789012345678900123456789001234567890
{attribute 'hide'}  EOF      : STRING[ 95]:= ';-- end of file ----------------------------------------------------------------';
{attribute 'hide'}  NEWLINE  : STRING[  3]:= '$0D$0A';
{attribute 'hide'}  DIVIDER  : STRING[ 95]:= ';-------------------------------------------------------------------------------';
{attribute 'hide'}  CREATED  : STRING[ 15]:= '; CREATED  : ';
{attribute 'hide'}  TD       : STRING[ 15]:= '; DATE     : ';
{attribute 'hide'}  ENCODING : STRING[ 19]:= '; ENCODING : UTF08';
{attribute 'hide'}  EMPTYLINE: STRING[  3]:= '; ';
{attribute 'hide'}  APPL     : STRING[ 15]:= '; APPL     : ';
{attribute 'hide'}  BUILD    : STRING[ 15]:= '; BUILD    : ';
{attribute 'hide'}  HOST     : STRING[ 15]:= '; HOST     : ';
{attribute 'hide'}  ADDR     : STRING[ 15]:= '; ADDR     : ';
{attribute 'hide'}  OPSYSTEM : STRING[ 15]:= '; SYSTEM   : ';
{attribute 'hide'}  RUNTIME  : STRING[ 19]:= '; RUNTIME  : TC';
{attribute 'hide'}  INFO     : STRING[ 15]:= '; INFO     : ';
{attribute 'hide'}  SIZE     : STRING[ 15]:= '; SIZE     : ';
{attribute 'hide'}  HEADER   : STRING[195]:= '; -- DATE & TIME ------- count -- level -- instance -------------------------- position ------- message ------- additional information ------';
END_VAR


(********************************************************************************************************************************)
(** calculate execution time ****************************************************************************************************)
_GetSystemTicks();
_StartSystemTick:= (         DWORD_TO_ULINT(_GetSystemTicks.cpuCntLoDW)
                     OR SHL( DWORD_TO_ULINT(_GetSystemTicks.cpuCntHiDW),  32 )  );




(********************************************************************************************************************************)
(** run all services ************************************************************************************************************)
_HddUsage();  // call here to use everywhere

M_RunHddUsage();
M_RunCheck();
M_RunWrite();
M_RunDelete();

IF (_MillisecondsLast = System.fbSystemTime.TIMESTR.wMilliseconds)
THEN
  _Diag_SystemTime:= _Diag_SystemTime + 1;

  (*-- trace it ---------------------------------------------------*)
  IF(_TaskCounter <> 0)
  THEN
// example: '11-000-0000-00-0,  system time not updated'
   ;(* _Text:= '';
    _Text:= CONCAT(_Text, F_AddDividerToSisString(SubsystemRegistry.SubsystemName) );
    _Text:= CONCAT(_Text, ',  system time not updated');
    Put( MsgType := E_DebugMsgType.WARNING,
         Instance:= ADR(_Instance),
         Text    := ADR(_Text)  );*)
  END_IF
END_IF

_MillisecondsLast:= System.fbSystemTime.TIMESTR.wMilliseconds;
_TaskCounter:= 0;




(********************************************************************************************************************************)
(** calculate execution time ****************************************************************************************************)
_GetSystemTicks();

_ExecutionNow:= (         DWORD_TO_ULINT(_GetSystemTicks.cpuCntLoDW)
                  OR SHL( DWORD_TO_ULINT(_GetSystemTicks.cpuCntHiDW),  32 )  );

_ExecutionDuration:= (_ExecutionNow - _StartSystemTick + 5) / 10;

_Statistics.MaxExecutionDuration:= MAX(_Statistics.MaxExecutionDuration, _ExecutionDuration);




(********************************************************************************************************************************)
(** done ************************************************************************************************************************)

// clears the internal fifo (all unwritten traces will be lost)
METHOD PUBLIC Clear

(********************************************************************************************************************************)
VAR_INPUT
END_VAR

(********************************************************************************************************************************)
VAR
  Index                 : WORD                             := 0;
  Entry                 : POINTER TO FB_TraceEntry         := 0;
END_VAR

(********************************************************************************************************************************)
(********************************************************************************************************************************)
_FifoFillLevel:= 0;
_FifoInput    := 0;
_FifoOutput   := 0;




(********************************************************************************************************************************)
(********************************************************************************************************************************)
Index:= 0;
WHILE (Index < FIFO_SIZE)
DO
  Entry:= _Fifo[Index];

  (*-- release memory -----------------------------------------------*)
  IF (Entry <> 0)
  THEN
    __DELETE(Entry);
  END_IF

  (*-- next ---------------------------------------------------------*)
  _Fifo[Index]:= 0;
  Index:= Index + 1;
END_WHILE




(********************************************************************************************************************************)
(** done ************************************************************************************************************************)
END_METHOD

// HI = writing/deleting enabled
{attribute 'monitoring' := 'call'}
PROPERTY PUBLIC Enable : BOOL
GET
Enable:= _Enable;
END_GET
SET
(********************************************************************************************************************************)
(** change? *********************************************************************************************************************)
IF (_Enable = Enable)
THEN
  RETURN;
END_IF

_Enable:= Enable;




(********************************************************************************************************************************)
(** done ************************************************************************************************************************)
END_SET
END_PROPERTY

{attribute 'hide'}
METHOD FB_exit : BOOL

(********************************************************************************************************************************)
VAR_INPUT
	bInCopyCode           : BOOL;  // if TRUE, the instance afterwards gets moved into the copy code (online change)
  (*----------------------------------------------------------------------------------------------------------------------------*)
END_VAR

(********************************************************************************************************************************)
(** release dynamically assigned memory *****************************************************************************************)
Clear();




(********************************************************************************************************************************)
(** done ************************************************************************************************************************)
END_METHOD

{attribute 'hide'}
METHOD FB_init : BOOL

(********************************************************************************************************************************)
VAR_INPUT
	bInitRetains          : BOOL; // if TRUE, the retain variables are initialized (warm start / cold start)
	bInCopyCode           : BOOL;  // if TRUE, the instance afterwards gets moved into the copy code (online change)
  (*----------------------------------------------------------------------------------------------------------------------------*)
END_VAR

(********************************************************************************************************************************)
VAR
END_VAR

(********************************************************************************************************************************)
(** remove 'QB2Jumpstart.JumpStart.' from instance path *************************************************************************)
F_InstancePathRemovals( DestStart     := ADR(_Instance),
                        DestEnd       := ADR(_Instance) + SIZEOF(_Instance),
                        RemoveLastPart:= FALSE );




(********************************************************************************************************************************)
(** done ************************************************************************************************************************)
END_METHOD

// folder to work within, folder must exist! (will only take effect when enabled is low)
{attribute 'monitoring' := 'call'}
PROPERTY PUBLIC Folder : A_TracePath
GET
Folder:= _Folder;
END_GET
SET
VAR
  Idx                   : WORD                             := 0;
  SepFound              : BOOL                             := FALSE;
  Finished              : BOOL                             := FALSE;
END_VAR
(********************************************************************************************************************************)
(** change? *********************************************************************************************************************)
IF (_Folder = Folder)
THEN
  RETURN;
END_IF

_Folder:= Folder;




(********************************************************************************************************************************)
(** change '\' to '/' and remove a trailing '/' if neccessary *******************************************************************)
Idx:= 0;
WHILE (Idx < SIZEOF(_Folder)  )
DO
  (*-- replace '\' with '/' -------------------------------------------------------------*)
  IF (_Folder[Idx] = 16#5C)  (* '\' *)
  THEN
    _Folder[Idx]:= 16#2F;   (* '/' *)
    SepFound:= TRUE;

  (*-- separation found '/' -------------------------------------------------------------*)
  ELSIF(_Folder[Idx] = 16#2F)   (* '/' *)
  THEN
    SepFound:= TRUE;

  (*-- fill rest of string with terminations --------------------------------------------*)
  ELSIF(Finished = TRUE)
  THEN
    (*-------------------------------------------*)
    _Folder[Idx]:= 16#00;

  (*-- string termination found ---------------------------------------------------------*)
  ELSIF(_Folder[Idx] = 16#00)
  THEN
    (*-- remove trailing '/' --------------------*)
    IF (SepFound = TRUE)
    THEN
      _Folder[Idx-1] := 16#00;
    END_IF
    (*-------------------------------------------*)
    Finished:= TRUE;
    SepFound:= FALSE;

  (*-- normal character -----------------------------------------------------------------*)
  ELSE
    SepFound:= FALSE;
  END_IF

  (*-- next -----------------------------------------------------------------------------*)
  Idx:= Idx + 1;
END_WHILE




(********************************************************************************************************************************)
(** done ************************************************************************************************************************)
END_SET
END_PROPERTY

// usage/free and total space of hdd
{attribute 'monitoring' := 'call'}
PROPERTY PUBLIC HddUsage : I_HddUsage
GET
HddUsage:= _HddUsage;
END_GET
END_PROPERTY

// builds the file name with index
METHOD PROTECTED M_BuildFileName

(********************************************************************************************************************************)
VAR
  DestStart             : POINTER TO BYTE                  := 0;     // start position to concat
  DestEnd               : POINTER TO BYTE                  := 0;     // buffer/string end
END_VAR

(********************************************************************************************************************************)
(********************************************************************************************************************************)
DestStart:= ADR(_WriteFileName);
DestEnd  := ADR(_WriteFileName) + SIZEOF(_WriteFileName);

(*-- application ---------------------------------------------------------------------------------------------------------------*)
DestStart:= F_StringCopy          ( DestStart:= DestStart,  DestEnd:= DestEnd,  Source    := ADR(_GetHostName.sHostName)  );

(*-- date ----------------------------------------------------------------------------------------------------------------------*)
DestStart:= F_StringCopy          ( DestStart:= DestStart,  DestEnd:= DestEnd,  Source    := ADR('_')  );
DestStart:= F_StringFromDatestruct( DestStart:= DestStart,  DestEnd:= DestEnd,  DateStruct:= _WriteDate );

(*-- index ---------------------------------------------------------------------------------------------------------------------*)
DestStart:= F_StringCopy          ( DestStart:= DestStart,  DestEnd:= DestEnd,  Source    := ADR('_')  );
DestStart:= F_StringFromWord      ( DestStart:= DestStart,  DestEnd:= DestEnd,  Value     := _FileIndex,  Length:= 4 );


(*-- file type -----------------------------------------------------------------------------------------------------------------*)
DestStart:= F_StringCopy          ( DestStart:= DestStart,  DestEnd:= DestEnd,  Source    := ADR('_Trace.txt')  );




(********************************************************************************************************************************)
(** done ************************************************************************************************************************)
END_METHOD

// created data to write, returns TRUE if trace date has changed
METHOD PROTECTED M_CreateData : BOOL

(********************************************************************************************************************************)
VAR
  MsgText               : STRING[31]                       := ''; 
  (*----------------------------------------------------------------------------------------------------------------------------*)
  DestStart             : POINTER TO BYTE                  := 0;
  DestWork              : POINTER TO BYTE                  := 0;
  DestEnd               : POINTER TO BYTE                  := 0;
  (*----------------------------------------------------------------------------------------------------------------------------*)
  EntryStart            : POINTER TO BYTE                  := 0;
  Entry                 : POINTER TO FB_TraceEntry         := 0;
  DateChanged           : BOOL                             := FALSE;
  Count                 : WORD                             := 0;
END_VAR

(********************************************************************************************************************************)
(********************************************************************************************************************************)
_DataLength:= 0;

DestStart:= ADR(_DataBuffer);
DestWork := ADR(_DataBuffer);
DestEnd  := ADR(_DataBuffer) + SIZEOF(_DataBuffer);

DateChanged:= FALSE;




(********************************************************************************************************************************)
(********************************************************************************************************************************)
Count:= 0;
WHILE(_FifoFillLevel <> 0)
DO
  (*-- get new entry --------------------------------------------------------------------*)
  Entry:= _Fifo[_FifoOutput];
  IF (Entry = 0)
  THEN
    EXIT;
  END_IF

  (*-- entry has already new date? ------------------------------------------------------*)
  IF (Entry^.IsEqualDate(_WriteDate) = FALSE)
  THEN
    DateChanged:= TRUE;
    EXIT;
  END_IF

  (*-- prepare line ---------------------------------------------------------------------*)
  MsgText:= TO_STRING(Entry^.MsgType);

  (*-- build line -----------------------------------------------------------------------*)
  EntryStart:= DestWork;
  DestWork:= F_StringFromDatestruct( DestStart:= DestWork,  DestEnd:= DestEnd,  DateStruct:= Entry^.DateTime  );
  DestWork:= F_StringCopy          ( DestStart:= DestWork,  DestEnd:= DestEnd,  Source    := ADR('  ')  );
  DestWork:= F_StringFromTimestruct( DestStart:= DestWork,  DestEnd:= DestEnd,  TimeStruct:= Entry^.DateTime,     ShowMs:= TRUE  );
  DestWork:= F_StringCopy          ( DestStart:= DestWork,  DestEnd:= DestEnd,  Source    := ADR(':  ')  );
  DestWork:= F_StringFromWord      ( DestStart:= DestWork,  DestEnd:= DestEnd,  Value     := Entry^.TaskCounter,  Length:= 0  );
  DestWork:= F_StringCopy          ( DestStart:= DestWork,  DestEnd:= DestEnd,  Source    := ADR(' = ')  );
  DestWork:= F_StringCopy          ( DestStart:= DestWork,  DestEnd:= DestEnd,  Source    := ADR(MsgText)  );
  DestWork:= F_StringCopy          ( DestStart:= DestWork,  DestEnd:= DestEnd,  Source    := ADR(',  ')  );
  DestWork:= F_StringCopy          ( DestStart:= DestWork,  DestEnd:= DestEnd,  Source    := Entry^.InstancePtr); 
  DestWork:= F_StringCopy          ( DestStart:= DestWork,  DestEnd:= DestEnd,  Source    := ADR(',  ')  );
  DestWork:= F_StringCopy          ( DestStart:= DestWork,  DestEnd:= DestEnd,  Source    := Entry^.TextPtr ); 
  DestWork:= F_StringCopy          ( DestStart:= DestWork,  DestEnd:= DestEnd,  Source    := ADR(NEWLINE)  );

  (*-- did not fit into write buffer (anymore) ------------------------------------------*)
  IF (DestWork >= DestEnd - 1)
  THEN
    DestWork:= EntryStart;
    EXIT;
  END_IF

  (*-- remove from fifo -----------------------------------------------------------------*)
  __DELETE(Entry);
  _Fifo[_FifoOutput]:= 0;

  (*-- next entry -> actualize fifo -----------------------------------------------------*)
  _FifoOutput:= _FifoOutput + 1;
  IF (_FifoOutput    >= FIFO_SIZE)  THEN  _FifoOutput:= 0;  END_IF
  IF (_FifoFillLevel > 0)           THEN  _FifoFillLevel:= _FifoFillLevel - 1;  END_IF

  (*-------------------------------------------------------------------------------------*)
  Count:= Count + 1;
END_WHILE

_Statistics.MaxDataItemsPerRow:= MAX(_Statistics.MaxDataItemsPerRow, Count);




(********************************************************************************************************************************)
(** calculate data length *******************************************************************************************************)
_DataLength:= (DestWork - DestStart);

_Statistics.MaxDataLength:= MAX(_Statistics.MaxDataLength, _DataLength);




(********************************************************************************************************************************)
(** done ************************************************************************************************************************)
M_CreateData:= DateChanged;
END_METHOD

// creates the eof file end
METHOD PROTECTED M_CreateEof

(********************************************************************************************************************************)
VAR
  DestStart             : POINTER TO BYTE                  := 0;
  DestWork              : POINTER TO BYTE                  := 0;
  DestEnd               : POINTER TO BYTE                  := 0;
END_VAR

(********************************************************************************************************************************)
(********************************************************************************************************************************)
_DataLength:= 0;

DestStart:= ADR(_DataBuffer);
DestWork := ADR(_DataBuffer);
DestEnd  := ADR(_DataBuffer) + SIZEOF(_DataBuffer);




(********************************************************************************************************************************)
(********************************************************************************************************************************)
DestWork:= F_StringCopy(DestStart:= DestWork, DestEnd:= DestEnd, Source:= ADR(NEWLINE)  );
DestWork:= F_StringCopy(DestStart:= DestWork, DestEnd:= DestEnd, Source:= ADR(EOF)      );
DestWork:= F_StringCopy(DestStart:= DestWork, DestEnd:= DestEnd, Source:= ADR(NEWLINE)  );
DestWork:= F_StringCopy(DestStart:= DestWork, DestEnd:= DestEnd, Source:= ADR(NEWLINE)  );




(********************************************************************************************************************************)
(** calculate data length *******************************************************************************************************)
_DataLength:= (DestWork - DestStart);

_Statistics.MaxDataLength:= MAX(_Statistics.MaxDataLength, _DataLength);




(********************************************************************************************************************************)
(** done ************************************************************************************************************************)
END_METHOD

// creates the file header for a new file
METHOD PROTECTED M_CreateHeader

(********************************************************************************************************************************)
VAR
  DestStart             : POINTER TO BYTE                  := 0;
  DestWork              : POINTER TO BYTE                  := 0;
  DestEnd               : POINTER TO BYTE                  := 0;
  (*----------------------------------------------------------------------------------------------------------------------------*)
  AdapterInfo           : ST_IpAdapterInfo;
  Idx                   : BYTE                             := 0;
END_VAR

(********************************************************************************************************************************)
(********************************************************************************************************************************)
_DataLength:= 0;

DestStart:= ADR(_DataBuffer);
DestWork := ADR(_DataBuffer);
DestEnd  := ADR(_DataBuffer) + SIZEOF(_DataBuffer);




(********************************************************************************************************************************)
(********************************************************************************************************************************)
(*-- ;-line --------------------------------------------------------------------------------------------------------------------*)
DestWork:= F_StringCopy( DestStart:= DestWork,  DestEnd:= DestEnd,  Source:= ADR(DIVIDER)  );
DestWork:= F_StringCopy( DestStart:= DestWork,  DestEnd:= DestEnd,  Source:= ADR(NEWLINE)  );


(*-- info line -----------------------------------------------------------------------------------------------------------------*)
DestWork:= F_StringCopy( DestStart:= DestWork,  DestEnd:= DestEnd,  Source:= ADR(CREATED)            );
DestWork:= F_StringCopy( DestStart:= DestWork,  DestEnd:= DestEnd,  Source:= ADR('FB_TraceHandler')  );
DestWork:= F_StringCopy( DestStart:= DestWork,  DestEnd:= DestEnd,  Source:= ADR('  ')               );
DestWork:= F_StringCopy( DestStart:= DestWork,  DestEnd:= DestEnd,  Source:= ADR('[b7lipim]')        );
DestWork:= F_StringCopy( DestStart:= DestWork,  DestEnd:= DestEnd,  Source:= ADR(NEWLINE)            );


(*-- Datum&Uhrzeit-Zeile bauen -------------------------------------------------------------------------------------------------*)
DestWork:= F_StringCopy          ( DestStart:= DestWork,  DestEnd:= DestEnd,  Source    := ADR(TD)          );
DestWork:= F_StringFromDatestruct( DestStart:= DestWork,  DestEnd:= DestEnd,  DateStruct:= System.fbSystemTime.TIMESTR  );
DestWork:= F_StringCopy          ( DestStart:= DestWork,  DestEnd:= DestEnd,  Source    := ADR('  ')        );
DestWork:= F_StringFromTimestruct( DestStart:= DestWork,  DestEnd:= DestEnd,  TimeStruct:= System.fbSystemTime.TIMESTR, ShowMs:= TRUE  );
DestWork:= F_StringCopy          ( DestStart:= DestWork,  DestEnd:= DestEnd,  Source    := ADR(NEWLINE)     );


(*-- Encoding Info -------------------------------------------------------------------------------------------------------------*)
DestWork:= F_StringCopy( DestStart:= DestWork,  DestEnd:= DestEnd,  Source:= ADR(ENCODING)  );
DestWork:= F_StringCopy( DestStart:= DestWork,  DestEnd:= DestEnd,  Source:= ADR(NEWLINE)   );


(*-- Applikation ---------------------------------------------------------------------------------------------------------------*)
DestWork:= F_StringCopy( DestStart:= DestWork,  DestEnd:= DestEnd,  Source:= ADR(EMPTYLINE) );
DestWork:= F_StringCopy( DestStart:= DestWork,  DestEnd:= DestEnd,  Source:= ADR(NEWLINE)   );
DestWork:= F_StringCopy( DestStart:= DestWork,  DestEnd:= DestEnd,  Source:= ADR(APPL)      );
DestWork:= F_StringCopy( DestStart:= DestWork,  DestEnd:= DestEnd,  Source:= ADR('??')      );
DestWork:= F_StringCopy( DestStart:= DestWork,  DestEnd:= DestEnd,  Source:= ADR('  ')      );
DestWork:= F_StringCopy( DestStart:= DestWork,  DestEnd:= DestEnd,  Source:= ADR('??')      );
DestWork:= F_StringCopy( DestStart:= DestWork,  DestEnd:= DestEnd,  Source:= ADR('  (')     );
DestWork:= F_StringCopy( DestStart:= DestWork,  DestEnd:= DestEnd,  Source:= ADR('??')      );
DestWork:= F_StringCopy( DestStart:= DestWork,  DestEnd:= DestEnd,  Source:= ADR(')' )      );
DestWork:= F_StringCopy( DestStart:= DestWork,  DestEnd:= DestEnd,  Source:= ADR(NEWLINE)   );


(*-- Build ---------------------------------------------------------------------------------------------------------------------*)


(*-- Host/Addr -----------------------------------------------------------------------------------------------------------------*)
DestWork:= F_StringCopy( DestStart:= DestWork,  DestEnd:= DestEnd,  Source:= ADR(EMPTYLINE) );
DestWork:= F_StringCopy( DestStart:= DestWork,  DestEnd:= DestEnd,  Source:= ADR(NEWLINE)   );
DestWork:= F_StringCopy( DestStart:= DestWork,  DestEnd:= DestEnd,  Source:= ADR(HOST)      );
DestWork:= F_StringCopy( DestStart:= DestWork,  DestEnd:= DestEnd,  Source:= ADR(_GetHostName.sHostName)  );
DestWork:= F_StringCopy( DestStart:= DestWork,  DestEnd:= DestEnd,  Source:= ADR(' @')      );
DestWork:= F_StringCopy( DestStart:= DestWork,  DestEnd:= DestEnd,  Source:= ADR(_GetDeviceIdentificationEx.stDevIdent.strAmsNetId) );
DestWork:= F_StringCopy( DestStart:= DestWork,  DestEnd:= DestEnd,  Source:= ADR(NEWLINE)   );

Idx:= 0;
WHILE(Idx <= Tc2_Utilities.MAX_LOCAL_ADAPTERS)
DO
  AdapterInfo:= _GetAdaptersInfo.arrAdapters[Idx];
  Idx:= Idx + 1;
  (*-- valid? ---------------------------------------------------------------------------*)
  IF(AdapterInfo.sIpAddr = '')         THEN  CONTINUE;  END_IF
  IF(AdapterInfo.sIpAddr = '0.0.0.0')  THEN  CONTINUE;  END_IF
  (*-------------------------------------------------------------------------------------*)
  DestWork:= F_StringCopy( DestStart:= DestWork,  DestEnd:= DestEnd,  Source:= ADR(ADDR)      );
  DestWork:= F_StringCopy( DestStart:= DestWork,  DestEnd:= DestEnd,  Source:= ADR(AdapterInfo.sIpAddr) );
  DestWork:= F_StringCopy( DestStart:= DestWork,  DestEnd:= DestEnd,  Source:= ADR('/') );
  DestWork:= F_StringCopy( DestStart:= DestWork,  DestEnd:= DestEnd,  Source:= ADR(AdapterInfo.sSubNet) );
  DestWork:= F_StringCopy( DestStart:= DestWork,  DestEnd:= DestEnd,  Source:= ADR('  {') );
  DestWork:= F_StringCopy( DestStart:= DestWork,  DestEnd:= DestEnd,  Source:= ADR(AdapterInfo.sDescription) );
  DestWork:= F_StringCopy( DestStart:= DestWork,  DestEnd:= DestEnd,  Source:= ADR('}') );
  (*-------------------------------------------------------------------------------------*)
  DestWork:= F_StringCopy( DestStart:= DestWork,  DestEnd:= DestEnd,  Source:= ADR(NEWLINE)   );
END_WHILE


(*-- System --------------------------------------------------------------------------------------------------------------------*)
DestWork:= F_StringCopy( DestStart:= DestWork,  DestEnd:= DestEnd,  Source:= ADR(EMPTYLINE) );
DestWork:= F_StringCopy( DestStart:= DestWork,  DestEnd:= DestEnd,  Source:= ADR(NEWLINE)   );
DestWork:= F_StringCopy( DestStart:= DestWork,  DestEnd:= DestEnd,  Source:= ADR(OPSYSTEM)  );
DestWork:= F_StringCopy( DestStart:= DestWork,  DestEnd:= DestEnd,  Source:= ADR(_GetDeviceIdentificationEx.stDevIdent.strImageOsName)    );
DestWork:= F_StringCopy( DestStart:= DestWork,  DestEnd:= DestEnd,  Source:= ADR('  {')    );
DestWork:= F_StringCopy( DestStart:= DestWork,  DestEnd:= DestEnd,  Source:= ADR(_GetDeviceIdentificationEx.stDevIdent.strImageOsVersion)    );
DestWork:= F_StringCopy( DestStart:= DestWork,  DestEnd:= DestEnd,  Source:= ADR('}')    );
DestWork:= F_StringCopy( DestStart:= DestWork,  DestEnd:= DestEnd,  Source:= ADR(NEWLINE)   );
DestWork:= F_StringCopy( DestStart:= DestWork,  DestEnd:= DestEnd,  Source:= ADR(RUNTIME)   );
DestWork:= F_StringCopy( DestStart:= DestWork,  DestEnd:= DestEnd,  Source:= ADR(_GetDeviceIdentificationEx.stDevIdent.strTwinCATVersion)    );
DestWork:= F_StringCopy( DestStart:= DestWork,  DestEnd:= DestEnd,  Source:= ADR('.')    );
DestWork:= F_StringCopy( DestStart:= DestWork,  DestEnd:= DestEnd,  Source:= ADR(_GetDeviceIdentificationEx.stDevIdent.strTwinCATRevision)   );
DestWork:= F_StringCopy( DestStart:= DestWork,  DestEnd:= DestEnd,  Source:= ADR('.')    );
DestWork:= F_StringCopy( DestStart:= DestWork,  DestEnd:= DestEnd,  Source:= ADR(_GetDeviceIdentificationEx.stDevIdent.strTwinCATBuild)      );
DestWork:= F_StringCopy( DestStart:= DestWork,  DestEnd:= DestEnd,  Source:= ADR(NEWLINE)         );



(*-- Info ----------------------------------------------------------------------------------------------------------------------*)
DestWork:= F_StringCopy    ( DestStart:= DestWork,  DestEnd:= DestEnd,  Source:= ADR(EMPTYLINE)       );
DestWork:= F_StringCopy    ( DestStart:= DestWork,  DestEnd:= DestEnd,  Source:= ADR(NEWLINE)         );
DestWork:= F_StringCopy    ( DestStart:= DestWork,  DestEnd:= DestEnd,  Source:= ADR(INFO)            );
DestWork:= F_StringCopy    ( DestStart:= DestWork,  DestEnd:= DestEnd,  Source:= ADR(_WriteFileName)  );
DestWork:= F_StringCopy    ( DestStart:= DestWork,  DestEnd:= DestEnd,  Source:= ADR(NEWLINE)         );
DestWork:= F_StringCopy    ( DestStart:= DestWork,  DestEnd:= DestEnd,  Source:= ADR(SIZE)            );
DestWork:= F_StringCopy    ( DestStart:= DestWork,  DestEnd:= DestEnd,  Source:= ADR('<= ')           );
DestWork:= F_StringFromWord( DestStart:= DestWork,  DestEnd:= DestEnd,  Value := _MaxFileSizeKB,  Length:= 0  );
DestWork:= F_StringCopy    ( DestStart:= DestWork,  DestEnd:= DestEnd,  Source:= ADR('kB')            );
DestWork:= F_StringCopy    ( DestStart:= DestWork,  DestEnd:= DestEnd,  Source:= ADR(NEWLINE)         );


(*-- ;-line --------------------------------------------------------------------------------------------------------------------*)
DestWork:= F_StringCopy( DestStart:= DestWork,  DestEnd:= DestEnd,  Source:= ADR(DIVIDER)  );
DestWork:= F_StringCopy( DestStart:= DestWork,  DestEnd:= DestEnd,  Source:= ADR(NEWLINE)  );




(********************************************************************************************************************************)
(** table header ****************************************************************************************************************)
DestWork:= F_StringCopy( DestStart:= DestWork,  DestEnd:= DestEnd,  Source:= ADR(NEWLINE)  );
DestWork:= F_StringCopy( DestStart:= DestWork,  DestEnd:= DestEnd,  Source:= ADR(NEWLINE)  );
DestWork:= F_StringCopy( DestStart:= DestWork,  DestEnd:= DestEnd,  Source:= ADR(HEADER)   );
DestWork:= F_StringCopy( DestStart:= DestWork,  DestEnd:= DestEnd,  Source:= ADR(NEWLINE)  );
DestWork:= F_StringCopy( DestStart:= DestWork,  DestEnd:= DestEnd,  Source:= ADR(NEWLINE)  );




(********************************************************************************************************************************)
(** calculate data length *******************************************************************************************************)
_DataLength:= (DestWork - DestStart);

_Statistics.MaxDataLength:= MAX(_Statistics.MaxDataLength, _DataLength);




(********************************************************************************************************************************)
(** done ************************************************************************************************************************)
END_METHOD

METHOD PROTECTED M_CreatePlcDivider

(********************************************************************************************************************************)
VAR
  DestStart             : POINTER TO BYTE                  := 0;
  DestWork              : POINTER TO BYTE                  := 0;
  DestEnd               : POINTER TO BYTE                  := 0;
  (*----------------------------------------------------------------------------------------------------------------------------*)
  DateString            : STRING[15]                       := '';
  TimeString            : STRING[15]                       := '';
  FileSize              : STRING[15]                       := '';
END_VAR

(********************************************************************************************************************************)
(********************************************************************************************************************************)
_DataLength:= 0;

DestStart:= ADR(_DataBuffer);
DestWork := ADR(_DataBuffer);
DestEnd  := ADR(_DataBuffer) + SIZEOF(_DataBuffer);




(********************************************************************************************************************************)
(********************************************************************************************************************************)
DestWork:= F_StringCopy(DestStart:= DestWork, DestEnd:= DestEnd, Source:= ADR(NEWLINE)  );
DestWork:= F_StringCopy(DestStart:= DestWork, DestEnd:= DestEnd, Source:= ADR(NEWLINE)  );




(********************************************************************************************************************************)
(** calculate data length *******************************************************************************************************)
_DataLength:= (DestWork - DestStart);

_Statistics.MaxDataLength:= MAX(_Statistics.MaxDataLength, _DataLength);




(********************************************************************************************************************************)
(** done ************************************************************************************************************************)
END_METHOD

// checks existence of working folder
METHOD PROTECTED M_RunCheck

(********************************************************************************************************************************)
VAR
END_VAR

(********************************************************************************************************************************)
(** initialization **************************************************************************************************************)
CASE(_CheckState) OF
E_TraceCheckStates.Initialization:
  (*-- ENTRY -------------------------------------------------------------------------------------------------------------------*)
    _CheckStateLast:= _CheckState;

  (*-- ACTION ------------------------------------------------------------------------------------------------------------------*)

  (*-- TRANSITION --------------------------------------------------------------------------------------------------------------*)
  _CheckState:= E_TraceCheckStates.Delay;




(********************************************************************************************************************************)
(** short delay *****************************************************************************************************************)
E_TraceCheckStates.Delay:
  (*-- ENTRY -------------------------------------------------------------------------------------------------------------------*)
  IF (_CheckStateLast <> _CheckState)
  THEN
    _CheckStateLast:= _CheckState;
    _CheckTime     := F_GetTimeMsTick();
    (*-----------------------------------------------------------------------------------*)
  END_IF

  (*-- ACTION ------------------------------------------------------------------------------------------------------------------*)

  (*-- TRANSITION --------------------------------------------------------------------------------------------------------------*)
  (*-- delay time over ------------------------------------------------------------------*)
  IF(F_GetTimeMsDiff(_CheckTime) >= T#1S)
  THEN
    _CheckState:= E_TraceCheckStates.Hostname;
  END_IF




(********************************************************************************************************************************)
(** retrieve hostname ***********************************************************************************************************)
E_TraceCheckStates.Hostname:
  (*-- ENTRY -------------------------------------------------------------------------------------------------------------------*)
  IF (_CheckStateLast <> _CheckState)
  THEN
    _CheckStateLast:= _CheckState;
    _CheckTime     := F_GetTimeMsTick();
    (*-----------------------------------------------------------------------------------*)
    _GetHostName(bExecute:= FALSE);
    _GetHostName.bExecute:= TRUE;
  END_IF

  (*-- ACTION ------------------------------------------------------------------------------------------------------------------*)
  _GetHostName();

  (*-- TRANSITION --------------------------------------------------------------------------------------------------------------*)
  IF (_GetHostName.bBusy = FALSE)
  THEN
    _CheckState:= E_TraceCheckStates.Adapters;
  END_IF




(********************************************************************************************************************************)
(** retrieve network adapters infos *********************************************************************************************)
E_TraceCheckStates.Adapters:
  (*-- ENTRY -------------------------------------------------------------------------------------------------------------------*)
  IF (_CheckStateLast <> _CheckState)
  THEN
    _CheckStateLast:= _CheckState;
    _CheckTime     := F_GetTimeMsTick();
    (*-----------------------------------------------------------------------------------*)
    _GetAdaptersInfo(bExecute:= FALSE);
    _GetAdaptersInfo.bExecute:= TRUE;
  END_IF

  (*-- ACTION ------------------------------------------------------------------------------------------------------------------*)
  _GetAdaptersInfo();

  (*-- TRANSITION --------------------------------------------------------------------------------------------------------------*)
  IF (_GetAdaptersInfo.bBusy = FALSE)
  THEN
    _CheckState:= E_TraceCheckStates.DeviceIdentification;
  END_IF




(********************************************************************************************************************************)
(** retrieve device identification **********************************************************************************************)
E_TraceCheckStates.DeviceIdentification:
  (*-- ENTRY -------------------------------------------------------------------------------------------------------------------*)
  IF (_CheckStateLast <> _CheckState)
  THEN
    _CheckStateLast:= _CheckState;
    _CheckTime     := F_GetTimeMsTick();
    (*-----------------------------------------------------------------------------------*)
    _GetDeviceIdentificationEx(bExecute:= FALSE);
    _GetDeviceIdentificationEx.bExecute:= TRUE;
  END_IF

  (*-- ACTION ------------------------------------------------------------------------------------------------------------------*)
  _GetDeviceIdentificationEx();

  (*-- TRANSITION --------------------------------------------------------------------------------------------------------------*)
  IF (_GetDeviceIdentificationEx.bBusy = FALSE)
  THEN
    _CheckState:= E_TraceCheckStates.Disabled;
  END_IF




(********************************************************************************************************************************)
(** fb disabled *****************************************************************************************************************)
E_TraceCheckStates.Disabled:
  (*-- ENTRY -------------------------------------------------------------------------------------------------------------------*)
  IF (_CheckStateLast <> _CheckState)
  THEN
    _CheckStateLast:= _CheckState;
    _CheckTime     := F_GetTimeMsTick();
    (*-----------------------------------------------------------------------------------*)
    _Active    := FALSE;
    _MainFolder:= '';
  END_IF

  (*-- ACTION ------------------------------------------------------------------------------------------------------------------*)

  (*-- TRANSITION --------------------------------------------------------------------------------------------------------------*)
  (*-- enabled --------------------------------------------------------------------------*)
  IF (_Enable = TRUE)
  THEN
    _MainFolder:= _Folder;
    (*-------------------------------------------*)
    _CheckState:= E_TraceCheckStates.HddCheck;
  END_IF




(********************************************************************************************************************************)
(** hdd usage read ******************************************************************************************************************************)
E_TraceCheckStates.HddCheck:
  (*-- ENTRY -------------------------------------------------------------------------------------------------------------------*)
  IF (_CheckStateLast <> _CheckState)
  THEN
    _CheckStateLast:= _CheckState;
    _CheckTime     := F_GetTimeMsTick();
    (*-----------------------------------------------------------------------------------*)
  END_IF

  (*-- ACTION ------------------------------------------------------------------------------------------------------------------*)

  (*-- TRANSITION --------------------------------------------------------------------------------------------------------------*)
  IF (F_GetTimeMsDiff(_HddUsageTime) >= T#5M)  THEN  _CheckState:= E_TraceCheckStates.HddUsage;
  ELSE                                               _CheckState:= E_TraceCheckStates.Start;
  END_IF




(********************************************************************************************************************************)
(** read hdd usage **************************************************************************************************************)
E_TraceCheckStates.HddUsage:
  (*-- ENTRY -------------------------------------------------------------------------------------------------------------------*)
  IF (_CheckStateLast <> _CheckState)
  THEN
    _CheckStateLast:= _CheckState;
    _CheckTime     := F_GetTimeMsTick();
    (*-----------------------------------------------------------------------------------*)
    _HddUsage.Start( Drive:= _MainFolder );  // use drive letter from main folder
    _HddUsageTime:= F_GetTimeMsTick();
  END_IF

  (*-- ACTION ------------------------------------------------------------------------------------------------------------------*)
    // _HddUsage() is called in main body to be used in other state machines as well

  (*-- TRANSITION --------------------------------------------------------------------------------------------------------------*)
  IF (_HddUsage.Busy = FALSE)
  THEN
    _HddUsageCount:= _HddUsageCount + 1;
    (*-------------------------------------------*)
    IF    (_HddUsage.Error           = TRUE)               THEN  _HddState:= E_TraceHddUsageStates.Unknown;
    ELSIF (_HddUsage.PercentageUsed >= HDD_ERROR_LEVEL)    THEN  _HddState:= E_TraceHddUsageStates.ErrorLevel;
    ELSIF (_HddUsage.PercentageUsed >= HDD_WARNING_LEVEL)  THEN  _HddState:= E_TraceHddUsageStates.WarningLevel;
    ELSE                                                         _HddState:= E_TraceHddUsageStates.EnoughFree;
    END_IF
    (*-------------------------------------------*)
    _CheckState:= E_TraceCheckStates.Start;
  END_IF




(********************************************************************************************************************************)
(** prepare work folder check ***************************************************************************************************)
E_TraceCheckStates.Start:
  (*-- ENTRY -------------------------------------------------------------------------------------------------------------------*)
  IF (_CheckStateLast <> _CheckState)
  THEN
    _CheckStateLast:= _CheckState;
    _CheckTime     := F_GetTimeMsTick();
    (*-----------------------------------------------------------------------------------*)
    _CheckWorkFolder.sNetID   := '';   // local
    _CheckWorkFolder.sPathName:= _MainFolder;   // without trailing '/'
    _CheckWorkFolder.eCmd     := Tc2_Utilities.E_EnumCmdType.eEnumCmd_First;
    _CheckWorkFolder.tTimeout := Tc2_System.DEFAULT_ADS_TIMEOUT;
  END_IF

  (*-- ACTION ------------------------------------------------------------------------------------------------------------------*)

  (*-- TRANSITION --------------------------------------------------------------------------------------------------------------*)
  _CheckState:= E_TraceCheckStates.Scan;




(********************************************************************************************************************************)
(** check folder exists *********************************************************************************************************)
E_TraceCheckStates.Scan:
  (*-- ENTRY -------------------------------------------------------------------------------------------------------------------*)
  IF (_CheckStateLast <> _CheckState)
  THEN
    _CheckStateLast:= _CheckState;
    _CheckTime     := F_GetTimeMsTick();
    (*-----------------------------------------------------------------------------------*)
{warning disable C0139}
    _CheckWorkFolder( bExecute:= FALSE );
    _CheckWorkFolder.sNetID   ;   // hier nicht beschreiben
    _CheckWorkFolder.sPathName;   // hier nicht beschreiben
    _CheckWorkFolder.eCmd     ;   // hier nicht beschreiben
    _CheckWorkFolder.bExecute := TRUE;
    _CheckWorkFolder.tTimeout ;   // hier nicht beschreiben
{warning restore C0139}
  END_IF

  (*-- ACTION ------------------------------------------------------------------------------------------------------------------*)
  _CheckWorkFolder();

  (*-- TRANSITION --------------------------------------------------------------------------------------------------------------*)
  IF (_CheckWorkFolder.bBusy = FALSE)
  THEN
    _CheckWorkFolder.eCmd:= Tc2_Utilities.E_EnumCmdType.eEnumCmd_Next;
    (*-- Fehler -------------------------------------------------------------------------*)
    IF (_CheckWorkFolder.bError = TRUE)
    THEN
      //ErrorText:= 'target unreachable: ' + _WorkNetId.Value
      _Active    := FALSE;
      _CheckState:= E_TraceCheckStates.Wait;
    (*-- end of directory reached -------------------------------------------------------*)
    ELSIF (_CheckWorkFolder.bEOE = TRUE)
    THEN
      //ErrorText:= 'path not found: ' + _FilePath
      _Active    := FALSE;
      _CheckState:= E_TraceCheckStates.Wait;
    (*-- found as directory -------------------------------------------------------------*)
    ELSIF (_CheckWorkFolder.stFindFile.fileAttributes.bDirectory = TRUE)
    THEN
      //ErrorText:= '';
      _Active    := TRUE;
      _CheckState:= E_TraceCheckStates.Cancel;
    (*-- keep searching -----------------------------------------------------------------*)
    ELSE
      _CheckStateLast:= E_TraceCheckStates.Initialization;  // Re-entry
    END_IF

  END_IF




(********************************************************************************************************************************)
(********************************************************************************************************************************)
E_TraceCheckStates.Cancel:
  (*-- ENTRY -------------------------------------------------------------------------------------------------------------------*)
  IF (_CheckStateLast <> _CheckState)
  THEN
    _CheckStateLast:= _CheckState;
    _CheckTime     := F_GetTimeMsTick();
    (*-----------------------------------------------------------------------------------*)
{warning disable C0139}
    _CheckWorkFolder( bExecute:= FALSE );
    _CheckWorkFolder.sNetID;      // hier nicht beschreiben
    _CheckWorkFolder.sPathName;   // hier nicht beschreiben
    _CheckWorkFolder.eCmd     := Tc2_Utilities.E_EnumCmdType.eEnumCmd_Abort;
    _CheckWorkFolder.bExecute := TRUE;
    _CheckWorkFolder.tTimeout ;   // hier nicht beschreiben
{warning restore C0139}
  END_IF

  (*-- ACTION ------------------------------------------------------------------------------------------------------------------*)
  _CheckWorkFolder();

  (*-- TRANSITION --------------------------------------------------------------------------------------------------------------*)
  IF (_CheckWorkFolder.bBusy = FALSE)
  THEN
    (*-- error --------------------------------------------------------------------------*)
    IF (_CheckWorkFolder.bError = TRUE)
    THEN
      //ErrorText:= 'target unreachable'
      _Active    := FALSE;
      _CheckState:= E_TraceCheckStates.Wait;
    (*-- end of directory reached -------------------------------------------------------*)
    ELSIF (_CheckWorkFolder.bEOE = TRUE)
    THEN
      _CheckState:= E_TraceCheckStates.Wait;
    (*-- keep cancelling ----------------------------------------------------------------*)
    ELSE
      _CheckStateLast:= E_TraceCheckStates.Initialization;  // Re-entry
    END_IF
  END_IF




(********************************************************************************************************************************)
(********************************************************************************************************************************)
E_TraceCheckStates.Wait:
  (*-- ENTRY -------------------------------------------------------------------------------------------------------------------*)
  IF (_CheckStateLast <> _CheckState)
  THEN
    _CheckStateLast:= _CheckState;
    _CheckTime     := F_GetTimeMsTick();
    (*-----------------------------------------------------------------------------------*)
  END_IF

  (*-- ACTION ------------------------------------------------------------------------------------------------------------------*)

  (*-- TRANSITION --------------------------------------------------------------------------------------------------------------*)
  (*-- disabled -------------------------------------------------------------------------*)
  IF (_Enable = FALSE)
  THEN
    _CheckState:= E_TraceCheckStates.Disabled;
  (*-- wait time over -------------------------------------------------------------------*)
  ELSIF(F_GetTimeMsDiff(_CheckTime) >= T#1S)
  THEN
    _CheckState:= E_TraceCheckStates.HddCheck;
  END_IF




(********************************************************************************************************************************)
(** unknown *********************************************************************************************************************)
ELSE
  _CheckState:= E_TraceCheckStates.Initialization;
END_CASE




(********************************************************************************************************************************)
(** done ************************************************************************************************************************)
END_METHOD

// deletes all files and folders older than specified
METHOD PROTECTED M_RunDelete

(********************************************************************************************************************************)
VAR
  FolderDate            : TIMESTRUCT;
  (*----------------------------------------------------------------------------------------------------------------------------*)
  SystemTimeTD          : DATE_AND_TIME                    := DT#1979-01-09-23:59:59;
  FolderTimeTD          : DATE_AND_TIME                    := DT#1979-01-09-23:59:59;
  Diff_Seconds          : LINT                             := 0;
  (*----------------------------------------------------------------------------------------------------------------------------*)
  DestStart             : POINTER TO BYTE                  := 0;     // start position to concat
  DestEnd               : POINTER TO BYTE                  := 0;     // buffer/string end
  Result                : BOOL                             := FALSE;
END_VAR

(********************************************************************************************************************************)
(** initialization **************************************************************************************************************)
CASE(_DeleteState) OF
E_TraceDeleteStates.Initialization:
  (*-- ENTRY -------------------------------------------------------------------------------------------------------------------*)
    _DeleteStateLast:= _DeleteState;

  (*-- ACTION ------------------------------------------------------------------------------------------------------------------*)

  (*-- TRANSITION --------------------------------------------------------------------------------------------------------------*)
  _DeleteState:= E_TraceDeleteStates.WaitFolder;




(********************************************************************************************************************************)
(** wait working folder *********************************************************************************************************)
E_TraceDeleteStates.WaitFolder:
  (*-- ENTRY -------------------------------------------------------------------------------------------------------------------*)
  IF (_DeleteStateLast <> _DeleteState)
  THEN
    _DeleteStateLast:= _DeleteState;
    _DeleteTime     := F_GetTimeMsTick();
    (*-----------------------------------------------------------------------------------*)
  END_IF

  (*-- ACTION ------------------------------------------------------------------------------------------------------------------*)

  (*-- TRANSITION --------------------------------------------------------------------------------------------------------------*)
  (*-- working folder exists ------------------------------------------------------------*)
  IF (_Active = TRUE)
  THEN
    _DeleteState:= E_TraceDeleteStates.WaitDelay;
  END_IF




(********************************************************************************************************************************)
(** wait awhile *****************************************************************************************************************)
E_TraceDeleteStates.WaitDelay:
  (*-- ENTRY -------------------------------------------------------------------------------------------------------------------*)
  IF (_DeleteStateLast <> _DeleteState)
  THEN
    _DeleteStateLast:= _DeleteState;
    _DeleteTime     := F_GetTimeMsTick();
    (*-----------------------------------------------------------------------------------*)
  END_IF

  (*-- ACTION ------------------------------------------------------------------------------------------------------------------*)

